TYPE st_ads_OneAxisMoveWithoutPosition :
STRUCT
	//Excute:BOOL;
	//Done:BOOL;
	//Busy  : BOOL;
	//Occupied : BOOL;
	
	HandShake					: st_HandshakeBase;
END_STRUCT
END_TYPE

(* stored: Version 1.1.0.1, ProductVersion 3.1.4024.13
   DUT st_ads_OneAxisMoveWithoutPosition: Id {9d089183-1ec2-4c88-922e-3f66e47ec6f2} *)
